// TIA Portal V17 export
// export: Created 2025-06-25T13:13:18.4120949Z, ExportSetting WithDefaults, DisplayName Totally Integrated Automation Portal, DisplayVersion V17 Update 8, DisplayName TIA Portal Openness, DisplayVersion V17 Update 8, DisplayName TIA Portal Version Control Interface, DisplayVersion V17, DisplayName STEP 7 Professional, DisplayVersion V17 Update 8, DisplayName STEP 7 Safety, DisplayVersion V17 Update 6, DisplayName WinCC Advanced, DisplayVersion V17 Update 8
FUNCTION_BLOCK "fbHoursCounter2"   // FB54, LAD
TITLE = Hours counter
{ S7_Optimized_Access := 'TRUE' }
AUTHOR : Heaten
VERSION : 0.1
// stored: AutoNumber true, IsIECCheckEnabled false, IsRetainMemResEnabled false, MemoryReserve 0, SetENOAutomatically false, UDAEnableTagReadback false
   VAR_INPUT
      bCLK : Bool;   // 1-second pulse
      bEnable : Bool;   // Enable counting
   END_VAR
   VAR_IN_OUT
      sTag : "stHoursCounter";
   END_VAR
   VAR
      Tick : Bool;
      Reset : Bool;
   END_VAR
   VAR_TEMP
      Clock : Bool;
   END_VAR
   VAR_TEMP   // added for the SCL form of the ladder/FBD networks
      _w1 : Bool;
   END_VAR
BEGIN

REGION Network 1: Clock bit
   // When bEnable = TRUE, increase the elapsed time count
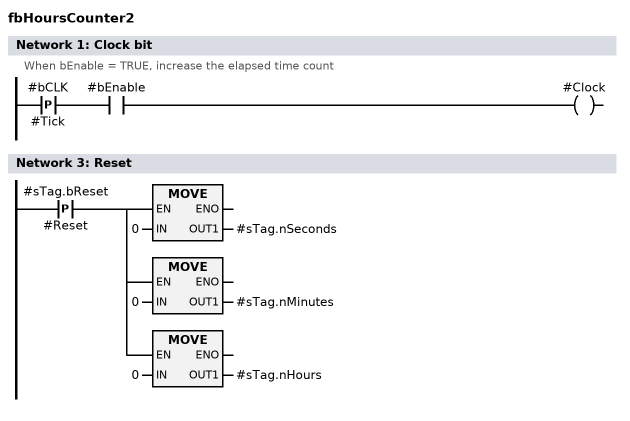
   RUNG wire#powerrail
      P_Contact(operand := #bCLK, bit := #Tick)
      Contact( #bEnable )
      Coil( #Clock )
   END_RUNG
   // the same network as SCL:
   #_w1 := #bCLK AND NOT #Tick;   // rising edge of #bCLK
   #Tick := #bCLK;
   #Clock := #_w1 AND #bEnable;
END_REGION

REGION Network 2 (SCL): Counting
   // Note: this is not automatically reset, should count up "forever" (approx equal to 490293 years).
   IF #Clock = TRUE THEN
       #sTag.nSeconds := #sTag.nSeconds + 1;
       IF #sTag.nSeconds > 59 THEN
           #sTag.nSeconds := 0;
           #sTag.nMinutes := #sTag.nMinutes + 1;
           IF #sTag.nMinutes > 59 THEN
               #sTag.nMinutes := 0;
               #sTag.nHours := #sTag.nHours + 1;
           END_IF;
       END_IF;
   END_IF;
END_REGION

REGION Network 3: Reset
   RUNG wire#powerrail
      P_Contact(operand := #sTag.bReset, bit := #Reset)
      wire#w1
      Move(in := 0, out1 => #sTag.nSeconds)
   END_RUNG
   RUNG wire#w1
      Move(in := 0, out1 => #sTag.nMinutes)
   END_RUNG
   RUNG wire#w1
      Move(in := 0, out1 => #sTag.nHours)
   END_RUNG
   // the same network as SCL:
   #_w1 := #sTag.bReset AND NOT #Reset;   // rising edge of #sTag.bReset
   #Reset := #sTag.bReset;
   IF #_w1 THEN
       #sTag.nSeconds := 0;
       #sTag.nMinutes := 0;
       #sTag.nHours := 0;
   END_IF;
END_REGION
END_FUNCTION_BLOCK
